(* CODESYS project PLC.library
   Company: Gema
   DefaultNamespace: RG
   Version: 0.1.1.1
   Placeholder: Rfid Reader
   Author: RG
   Description: Functionlity of RFID Reader
   Title: Rfid Reader

Project tree, tasks and I/O mapping:
  libraries: RFID universal data interface TwinCAT, 1.0.0.0 (Turck); Tc2_Standard, 3.3.3.0 (Beckhoff Automation GmbH); Tc2_System, 3.4.26.0 (Beckhoff Automation GmbH); Tc2_Utilities, 3.3.54.0 (Beckhoff Automation GmbH); Tc3_Module, 3.3.21.0 (Beckhoff Automation GmbH); TcoCore, 0.10.0.30 (Vortex.Library); TcoData, 0.10.0.31 (Vortex.Library); TcoDrivesBeckhoff, 0.10.0.31 (Vortex.Library); TcoElements, 0.10.0.31 (Vortex.Library); TcoPneumatics, 0.10.0.31 (Vortex.Library); TcUnit, * (www.tcunit.org)
  DUTs/
  GVLs/
  POUs/
  Rfid/
    Tasks/
      function block ReadUidTask [ST]: FB_init, OnDone, OnStart, Restore
    interface IRfidTasks: ReadUid
    function block RfidHead [ST]: ReadUidMethod, ReadUidTask, FB_init, Restore, ServiceMode
  Test/
    Context/
      function block AppContext [ST]: Main
      function block MainStation [ST]
      program PRG_TEST [ST]
    function block RfidHead_Test [ST]: ExecuteReadUid_ExpectUidAsStringStatusDone, FB_init
  Version/
    global variables Global_Version
  VISUs/
*)

// Version/Global_Version
{attribute 'TcGenerated'}
{attribute 'no-analysis'}
{attribute 'linkalways'}
// This function has been automatically generated from the project information.
VAR_GLOBAL CONSTANT
	{attribute 'const_non_replaced'}
	stLibVersion_Rfid_Reader : ST_LibVersion := (iMajor := 0, iMinor := 1, iBuild := 1, iRevision := 1, nFlags := 0, sVersion := '0.1.1.1');
END_VAR

// Rfid/Tasks/ReadUidTask
FUNCTION_BLOCK ReadUidTask EXTENDS TcoCore.TcoTask
VAR_IN_OUT
    turckRfid : RFID_FB_U.FB_Compact;
END_VAR
VAR_INPUT
    ActionDesc : STRING(25);
END_VAR
VAR_OUTPUT
    sUid : Tc2_System.T_MaxString;
END_VAR

VAR
    _stringBuilder : TcoCore.StringBuilder;
    _state : INT;
    _coding : ARRAY[0..7] OF BYTE;
    _index : INT;
    _hex : Tc2_System.T_MaxString := '16# ';
    _delay : TIME := T#1MS;
    _uidDataLength : UINT := 8;
    myReadData : ARRAY[0..127] OF POINTER TO BYTE;

END_VAR

IF (THIS^.Execute()) THEN
    CASE _state OF

        10:
            // Tag vorhanden
            IF NOT turckRfid.xTP THEN
                THIS^.Messenger.Error(
                    _stringBuilder.Append(ActionDesc)
                        .Append('Tag nicht vorhanden bei Leseversuch')
                        .ToString()
                );

                ThrowWhen(TRUE);
            ELSE
                _state := 20;
            END_IF
        20:
            //Command setzen
            turckRfid.eCommand := command.INVENTORY;
            //            turckRfid.uiDataLength := _uidDataLength;
            _state := 30;
        30:
            // Start der Operation
            turckRfid.xExecute := TRUE;
            sUid := '';

            _state := 40;
        40:
            // Warte auf Ende Operation
            IF turckRfid.xError THEN
                ;
            ELSIF turckRfid.xDone THEN
                FOR _index := 0 TO UINT_TO_INT(_uidDataLength - 1) DO
                    myReadData[_index] :=
                        (THIS^.turckRfid.pReadDataMapping + _index * SIZEOF(BYTE));
                    sUid := Concat(
                        sUid,
                        BYTE_TO_HEXSTR(in:=myReadData[_index]^, iPrecision:=2, bLoCase:=FALSE)
                    );
                END_FOR

                THIS^.DoneWhen(turckRfid.xDone);
                THIS^.Messenger.Info('Lesen UID erfolgreich');
                _state := 0;
            END_IF
    END_CASE
END_IF

METHOD PUBLIC FB_init : BOOL
VAR_INPUT
    bInitRetains : BOOL; // if TRUE, the retain variables are initialized (warm start / cold start)
    bInCopyCode : BOOL; // if TRUE, the instance afterwards gets moved into the copy code (online change)
    ParentObject : ITcoObject;
END_VAR
// This is not clear to me... I from time to time the consumer code does not see 'FB_init' of 'TcoObject', that's why overridden here with super call...
SUPER^.FB_init(bInitRetains, bInCopyCode, ParentObject);
END_METHOD

(*~
    <docu>
        <summary>
            Executes when task reaches the ```Done``` state .
        </summary>
    </docu>
~*)
METHOD PROTECTED OnDone
turckRfid.xExecute := false;
END_METHOD

(*~
    <docu>
        <summary>
            Executes ones when the task starts (at the moment of transition from the ```Requested``` state into the ```Busy``` state).
        </summary>
    </docu>
~*)
METHOD PROTECTED OnStart
turckRfid.eCommand := RFID_FB_U.COMMAND.IDLE;
turckRfid.xExecute := FALSE;
turckRfid.xAbort := FALSE;
_state := 10;
END_METHOD

(*~
    <docu>
        <summary>
            Restores this instance to the Ready state. Can be called explicitly or from within one of the restore mechanisms.
            <para>
                See also <see cref="PlcDocu.TcoCore.TcoTask.AutoRestorable()"/>
            </para>
        </summary>
    </docu>
~*)
METHOD Restore : ITcoRestorable
turckRfid.eCommand := RFID_FB_U.COMMAND.IDLE;
turckRfid.xExecute := FALSE;
turckRfid.xAbort := true;
END_METHOD

END_FUNCTION_BLOCK

// Rfid/IRfidTasks
INTERFACE IRfidTasks

METHOD ReadUid : BOOL
VAR_INPUT
END_VAR
END_METHOD

END_INTERFACE

// Rfid/RfidHead
FUNCTION_BLOCK RfidHead EXTENDS TcoCore.TcoComponent
VAR_OUTPUT
    sUId : T_MaxString;
END_VAR
VAR
    //Instantiate the function block (FB_BusMode)
    turckRfid : RFID_FB_U.FB_Compact;

    // Working buffers for the read and write data
    myReadData : ARRAY[0..127] OF BYTE;
    myWriteData : ARRAY[0..127] OF BYTE;

    // Create mapping to the I/O data of the corresponding channel
    stCompactModeRfidDiagMap AT %I* : ChannelDiag_t;

    stCompactModeInputMap AT %I* : RFID_FB_U.CompactInput_t;
    stCompactModeOutputMap AT %Q* : RFID_FB_U.CompactOutput_t;
    // The Rx & Tx data mapping shown below is for example purposes only.
    // The actual array size can be 8,16,32,64 or 128 depending on slot configuration of the TBEC-LL-4RFID-8DXP box in the IO tree
    abyRxDataMapCompactMode AT %I* : ARRAY[0..127] OF BYTE;
    abyTxDataMapCompactMode AT %Q* : ARRAY[0..127] OF BYTE;

    state : (Idle,
        Inventory,
        ReadBlock,
        WriteBlock,
        LockBlock,
        Abort,
        Error);
END_VAR
VAR
    _udiTimeOut : UDINT;
    _readUidTask : ReadUidTask(THIS^);

END_VAR

turckRfid(
    xExecute:=,
    rStatusMapping:=stCompactModeInputMap,
    rControlMapping:=stCompactModeOutputMap,
    pReadDataMapping:=abyRxDataMapCompactMode,
    pWriteDataMapping:=abyTxDataMapCompactMode,
    pDataTx:=myWriteData,
    pDataRx:=myReadData
);

_readUidTask(turckRfid:=turckRfid, ActionDesc:='<#ReadUid#>', sUid=>sUId);

//wichtig beim schreiben, length mitgeben
//bei Locked muss TO eingetellt werden, sonst kein Fehler
Case state of
    Idle:
    //        turckRfid.eCommand := RFID_FB_U.COMMAND.IDLE;
    //        turckRfid.xExecute := FALSE;
    //        turckRfid.xAbort := FALSE;

    Inventory:
        turckRfid.eCommand := RFID_FB_U.COMMAND.INVENTORY;
        turckRfid.xExecute := TRUE;

        IF turckRfid.xError THEN
            state := Error;
        ELSIF turckRfid.xDone THEN
            state := Idle;
            //            turckRfid.pDataTx := ADR(myWriteData);
            //            turckRfid.pDataRx := ADR(myReadData);
        END_IF

    ReadBlock:
        turckRfid.eCommand := RFID_FB_U.COMMAND.READ;
        turckRfid.uiDataLength := 4;
        turckRfid.xExecute := TRUE;

        IF turckRfid.xError THEN
            state := Error;
        ELSIF turckRfid.xDone THEN
            state := Idle;
            turckRfid.pDataTx := ADR(myWriteData);
            turckRfid.pDataRx := ADR(myReadData);
        END_IF

    WriteBlock:
        turckRfid.eCommand := RFID_FB_U.COMMAND.WRITE_AND_VERIFY;
        turckRfid.uiDataLength := 4;
        turckRfid.xExecute := TRUE;

        IF turckRfid.xError THEN
            state := Error;
        ELSIF turckRfid.xDone THEN
            state := Idle;
            turckRfid.pDataTx := ADR(myWriteData);
            turckRfid.pDataRx := ADR(myReadData);
        END_IF

    LockBlock:
        turckRfid.eCommand := RFID_FB_U.COMMAND.SET_PERMA_LOCK;
        turckRfid.xExecute := TRUE;

        IF turckRfid.xError THEN
            state := Error;
        ELSIF turckRfid.xDone THEN
            state := Idle;
            turckRfid.pDataTx := ADR(myWriteData);
            turckRfid.pDataRx := ADR(myReadData);
        END_IF

    Abort:
        turckRfid.eCommand := RFID_FB_U.COMMAND.IDLE;
        turckRfid.xAbort := TRUE;

    Error:
        ;
END_CASE

METHOD ReadUidMethod : TcoCore.ITcoTaskStatus
VAR_INPUT
END_VAR
IF (ReadUidTask <> 0) THEN
    ReadUidMethod := ReadUidTask.Invoke();
END_IF
END_METHOD

PROPERTY ReadUidTask : TcoCore.ITcoTask
GET
ReadUidTask := _readUidTask;
END_GET
END_PROPERTY

METHOD FB_init : BOOL
VAR_INPUT
    bInitRetains : BOOL; // if TRUE, the retain variables are initialized (warm start / cold start)
    bInCopyCode : BOOL; // if TRUE, the instance afterwards gets moved into the copy code (online change)
    ParentObject : ITcoObject;
    udiTimeOut : TIME;
END_VAR
VAR
    microToMillis : UDINT := 1000;
END_VAR
// This is not clear to me... I from time to time the consumer code does not see 'FB_init' of 'TcoObject', that's why overridden here with super call...
SUPER^.FB_init(bInitRetains, bInCopyCode, ParentObject);
this^._udiTimeOut := time_to_udint(udiTimeOut) * microToMillis;
END_METHOD

(*~
    <docu>
        <summary>
            Restore all tasks of this instance into initial state.
        </summary>
    </docu>
~*)
METHOD Restore : ITcoRestorable
//IF (AutoReadDataTask <> 0) THEN
//    AutoReadDataTask.Restore();
//END_IF;

//IF (AutoWriteDataTask <> 0) THEN
//    AutoWriteDataTask.Restore();
//END_IF;

//IF (ReadUidTask <> 0) THEN
//    ReadUidTask.Restore();
//END_IF;

//IF (ReadCodingTask <> 0) THEN
//    ReadCodingTask.Restore();
//END_IF;

//IF (WriteCodingTask <> 0) THEN
//	WriteCodingTask.Abort();
//    WriteCodingTask.Restore();
//END_IF;
END_METHOD

METHOD PROTECTED ServiceMode
END_METHOD

END_FUNCTION_BLOCK

// Test/Context/AppContext
FUNCTION_BLOCK AppContext EXTENDS TcoCore.TcoContext
VAR
    _mainStation : MainStation(THIS^);

    {attribute addProperty Name "Versionsnummer Plc"}
    _sVersion : STRING(23);
    //~
    _stProgramVersion : ST_LibVersion;
    //~

END_VAR

(*~
    <docu>
        <summary>
            Main method of the TcoContext. This is the entry point of any control logic that belongs to this context.
            The call of this method is ensured by calling the <c>InstanceName.Run()</c> method, and it must not be called explicitly.
            This method is abstract, and it must be overridden in derived block.
        </summary>
    </docu>
~*)
METHOD PROTECTED Main
_mainStation();
END_METHOD

END_FUNCTION_BLOCK

// Test/Context/MainStation
FUNCTION_BLOCK MainStation EXTENDS TcoCore.TcoObject
VAR
    turckRfidHead : RfidHead(THIS^, T#1MS);
    sUId          : T_MaxString;
    _uid          : BOOL;
END_VAR

turckRfidHead();

IF _uid THEN
    turckRfidHead.ReadUidMethod();
    _uid := FALSE;
END_IF

IF turckRfidHead.ReadUidTask.Done then
    sUId := turckRfidHead.sUId;
END_IF

END_FUNCTION_BLOCK

// Test/Context/PRG_TEST
PROGRAM PRG_TEST
VAR
    _testSuite : AppContext;
END_VAR

_testSuite.Run();
_testSuite.RtcSynchronize(true, '', 60);

END_PROGRAM

// Test/RfidHead_Test
FUNCTION_BLOCK RfidHead_Test EXTENDS TcUnit.FB_TestSuite

ExecuteReadUid_ExpectUidAsStringStatusDone();

METHOD PRIVATE ExecuteReadUid_ExpectUidAsStringStatusDone
VAR_INST
    turckRfidHead : RfidHead(THIS^, T#1MS);
    sUId          : T_MaxString;
    _uid          : BOOL;
END_VAR
TcUnit.TEST('ExecuteReadUid_ExpectUidAsStringStatusDone');
turckRfidHead();

IF _uid THEN
    turckRfidHead.ReadUidMethod();
    _uid := FALSE;
END_IF

IF turckRfidHead.ReadUidTask.Done then
    sUId := turckRfidHead.sUId;
END_IF

TcUnit.TEST_FINISHED();
END_METHOD

METHOD FB_init : BOOL
VAR_INPUT
    bInitRetains : BOOL; // if TRUE, the retain variables are initialized (warm start / cold start)
    bInCopyCode : BOOL; // if TRUE, the instance afterwards gets moved into the copy code (online change)
    ParentObject : ITcoObject;
    udiTimeOut : TIME;
END_VAR
VAR
    microToMillis : UDINT := 1000;
END_VAR
// This is not clear to me... I from time to time the consumer code does not see 'FB_init' of 'TcoObject', that's why overridden here with super call...
SUPER^.FB_init(bInitRetains, bInCopyCode, ParentObject);
this^._udiTimeOut := time_to_udint(udiTimeOut) * microToMillis;
END_METHOD

END_FUNCTION_BLOCK
